// TIA Portal V16 export
// export: Created 2024-12-03T15:41:39.3623529Z, ExportSetting WithDefaults, DisplayName Totally Integrated Automation Portal, DisplayVersion V16 Update 6, DisplayName TIA Portal Version Control Interface, DisplayVersion V16 Update 2, DisplayName TIA Portal Openness, DisplayVersion V16 Update 6, DisplayName TIA Portal Teamcenter Gateway, DisplayVersion V16, DisplayName SINAMICS Startdrive Advanced, DisplayVersion V16 Update 5, DisplayName SINAMICS Startdrive G130, G150, S120, S150, SINAMICS MV, S210, DisplayVersion V16 Update 5, DisplayName SINAMICS Startdrive G110M, G120, G120C, G120D, G120P, G115D, DisplayVersion V16 Update 5, DisplayName STEP 7 Professional, DisplayVersion V16 Update 6, DisplayName STEP 7 Safety, DisplayVersion V16, DisplayName WinCC Advanced / Unified PC, DisplayVersion V16 Update 6
FUNCTION_BLOCK "InputReaderDrive_FB"   // FB7, SCL
{ S7_Optimized_Access := 'TRUE' }
VERSION : 0.1
// stored: AutoNumber true, IsIECCheckEnabled false, IsRetainMemResEnabled false, MemoryReserve 100, SetENOAutomatically false, UDAEnableTagReadback false
   VAR
      FTC_DRV_101_1_I1 : "SmartBool";
      FTC_DRV_101_1_I2 : "SmartBool";
      FTC_DRV_101_1_I3 : "SmartBool";
      FTC_DRV_101_1_I4 : "SmartBool";
      FTC_SKU_101_I1 { S7_SetPoint := 'True'} : "SmartBool";
      FTC_SKU_101_I2 { S7_SetPoint := 'True'} : "SmartBool";
   END_VAR
BEGIN
   REGION DRV_101_1 

       #FTC_DRV_101_1_I1(I_Sensor := NOT "I_DRV_101_1".DigitalInputs.Input_1,
                        O_data => "Inputs_DB".FTC_DRV_101_1_I1);

       #FTC_DRV_101_1_I2(I_Sensor := NOT "I_DRV_101_1".DigitalInputs.Input_2,
                        O_data => "Inputs_DB".FTC_DRV_101_1_I2);

       #FTC_DRV_101_1_I3(I_Sensor := NOT "I_DRV_101_1".DigitalInputs.Input_3,
                        O_data => "Inputs_DB".FTC_DRV_101_1_I3);

       #FTC_DRV_101_1_I4(I_Sensor := NOT "I_DRV_101_1".DigitalInputs.Input_4,
                        O_data => "Inputs_DB".FTC_DRV_101_1_I4);

   END_REGION

   REGION SKU_101 

       #FTC_SKU_101_I1(I_Sensor := NOT "I_SKU_101".Input_1,
                      O_data => "Inputs_DB".FTC_SKU_101_I1);

       #FTC_SKU_101_I2(I_Sensor := NOT "I_SKU_101".Input_2,
                      O_data => "Inputs_DB".FTC_SKU_101_I2);

   END_REGION
END_FUNCTION_BLOCK
